(* IEC 61131-3 sources: beckhoffAutomationInterface/ST/Shark/Lib/Sequences (part 2) *)

(* ---- FB_SequenceTester.st ---- *)
(*
FB_SequenceTester — Shared test harness for sequence development.

Calls FB_SequenceOrchestrator methods directly via a REFERENCE.
Held inside a thin PROGRAM wrapper in each machine's App folder.

USAGE (thin PROGRAM wrapper pattern):
  PROGRAM PRG_SequenceTester
  VAR
      fbTester : FB_SequenceTester;
  END_VAR
      fbTester();
  // Configure: PRG_SequenceTester.Configure(refOrchestrator := PRG_Sequence.fbOrchestrator)

HOW TO TEST:
1. Set eCommand to desired command (e.g., E_Command.StartBubblerFlow)
2. Configure the corresponding parameter structure if needed
3. Set bStart := TRUE (pulse — auto-clears on rising edge)
4. Monitor sStatus, bBusy, bDone, bError, rProgress
*)
FUNCTION_BLOCK FB_SequenceTester
VAR
    // User interface — command triggers (pulse TRUE to execute)
    bStart   : BOOL;
    bStop    : BOOL;
    bReset   : BOOL;
    eCommand : E_Command := E_Command.StartBubblerFlow;

    // Parameter structures (pre-configured with realistic defaults)
    stBubblerFlowParams     : ST_CmdStartBubblerFlow := (
        side := 1,
        bubblerIndex := 1,
        flowRate := 15.0,
        hotManifoldOperatingPressure := 1.4,
        hotManifoldPressureTimeout := 600000,
        coldManifoldOperatingPressure := 1.4,
        coldManifoldPressureTimeout := 600000,
        MFCStabilizeTimeout := 60000,
        MFCFlowRateTolerance := 5.0,
        maxDepressurizingAttempts := 3
    );

    stStopBubblerFlowParams : ST_CmdStopBubblerFlow := (
        side := 1
    );

    stPurgeParams           : ST_CmdPurge := (
        mode := 1,
        side := 1,
        bubbler := 1,
        inertGasFlow := 300.0,
        purgeGasFlow := 25.0,
        purgeHighPressureLimit := 1.70,
        purgeLowPressureLimit := 0.75,
        hotManifoldOperatingPressure := 1.4,
        highPressureTimeout := 600000,
        lowPressureTimeout := 60000,
        coldManifoldPurgeCycles := 5,
        hotManifoldPurgeCycles := 5,
        purgeLinePurgeCycles := 5,
        umbilicalPurgeCycles := 5,
        umbilicalFlushTime := 60000,
        stabilisationDelay := 35000
    );

    stHeatingParams         : ST_CmdSetTemperatureGradient := (
        reactantCombiner := 60.0,
        precursorCombiner := 60.0,
        headTemp := 100.0,
        enableMode := 0
    );

    stChuckParams           : ST_CmdSetChuckZone := (
        holdSample := TRUE,
        size := 200,
        fPressureThreshold := 0.75,
        tPressureTimeout := 60000
    );

    stSpotDepositionParams  : ST_CmdSpotDeposition := (
        nDepositionCycles := 5,
        fPrecursorFlowRate := 20.0,
        fReactantFlowRate := 20.0,
        fInertMaxPurgeFlow := 250.0,
        fInertMinPurgeFlow := 100.0,
        nPrecursorBubblerIndex := 1,
        nReactantBubblerIndex := 1,
        fDistributorOperatingPressure := 2.0,
        fCombinerOperatingPressure := 1.3,
        fPressureTolerance := 5.0,
        tReactantExposureTime := 3000,
        tPrecursorExposureTime := 3000,
        tInertPurgeTime := 10000,
        tFinalPurgeTime := 30000
    );

    stLeakTestParams        : ST_CmdBubblerLeakTest := (
        side := 1,
        bubblerIndex := 1,
        leakThreshold := 0.5,
        testDuration := 300000,
        stabilizationTime := 60000,
        fillPressure := 2.5,
        testFlowRate := 20.0,
        pressureTimeout := 600000,
        pressureTolerance := 5.0,
        normalPressure := 1.4,
        depressurizeTarget := 0.5,
        normalizationFlow := 20.0
    );

    // Status output
    sStatus              : STRING(255) := 'Not configured';
    bBusy                : BOOL;
    bDone                : BOOL;
    bError               : BOOL;
    rProgress            : REAL;
    stStatus             : ST_SequenceStatus;
    stLastError          : ST_Error;
    sLastCommandResult   : STRING(255);
    bLastCommandAccepted : BOOL;

    // Debug counters
    nCycleCount   : UDINT := 0;
    nCommandCount : UDINT := 0;
    bTriggerFired : BOOL;
END_VAR
VAR
    _refOrchestrator : REFERENCE TO FB_SequenceOrchestrator;
    _bConfigured     : BOOL := FALSE;
    _rtStart         : R_TRIG;
    _rtStop          : R_TRIG;
    _rtReset         : R_TRIG;
    _sPrevStatusMsg  : STRING(255);
END_VAR

    nCycleCount   := nCycleCount + 1;
    bTriggerFired := FALSE;

    _rtStart(CLK := bStart);
    _rtStop(CLK  := bStop);
    _rtReset(CLK := bReset);

    IF NOT _bConfigured OR NOT __ISVALIDREF(_refOrchestrator) THEN
        sStatus := 'Waiting for orchestrator...';
        RETURN;
    END_IF

    IF _rtStop.Q THEN
        bStop         := FALSE;
        bTriggerFired := TRUE;
        bLastCommandAccepted := _refOrchestrator.SystemStop();
        sLastCommandResult := SEL(bLastCommandAccepted, 'SystemStop REJECTED', 'SystemStop accepted');
        nCommandCount := nCommandCount + 1;
    END_IF

    IF _rtReset.Q THEN
        bReset        := FALSE;
        bTriggerFired := TRUE;
        bLastCommandAccepted := _refOrchestrator.ErrorAcknowledge();
        sLastCommandResult := SEL(bLastCommandAccepted,
            'ErrorAcknowledge REJECTED (not in error state)',
            'ErrorAcknowledge accepted');
        nCommandCount := nCommandCount + 1;
    END_IF

    IF _rtStart.Q THEN
        bStart        := FALSE;
        bTriggerFired := TRUE;
        _ExecuteCommand();
        nCommandCount := nCommandCount + 1;
    END_IF

    stStatus    := _refOrchestrator.GetStatus();
    bBusy       := stStatus.bBusy;
    bDone       := stStatus.bDone;
    bError      := stStatus.bError;
    rProgress   := stStatus.rProgress;
    stLastError := stStatus.stLastError;

    IF bBusy THEN
        IF stStatus.sStatusMessage <> _sPrevStatusMsg THEN
            sStatus         := CONCAT('BUSY: ', stStatus.sStatusMessage);
            _sPrevStatusMsg := stStatus.sStatusMessage;
        END_IF
    ELSIF bError THEN
        IF stStatus.sStatusMessage <> _sPrevStatusMsg THEN
            sStatus         := CONCAT('ERROR: ', stStatus.sStatusMessage);
            _sPrevStatusMsg := stStatus.sStatusMessage;
        END_IF
    ELSIF bDone THEN
        IF stStatus.sStatusMessage <> _sPrevStatusMsg THEN
            sStatus         := CONCAT('DONE: ', stStatus.sStatusMessage);
            _sPrevStatusMsg := stStatus.sStatusMessage;
        END_IF
    ELSE
        sStatus         := SEL(sLastCommandResult = '', 'Ready', sLastCommandResult);
        _sPrevStatusMsg := '';
    END_IF

END_FUNCTION_BLOCK

// =============================================================================
// PUBLIC API
// =============================================================================

METHOD PUBLIC Configure : BOOL
VAR_INPUT
    refOrchestrator : REFERENCE TO FB_SequenceOrchestrator;
END_VAR
    IF NOT __ISVALIDREF(refOrchestrator) THEN RETURN; END_IF
    _refOrchestrator REF= refOrchestrator;
    _bConfigured     := TRUE;
    sStatus          := 'Ready';
    sLastCommandResult := '';
    Configure        := TRUE;
END_METHOD

// =============================================================================
// PRIVATE
// =============================================================================

METHOD PRIVATE _ExecuteCommand
VAR
    bSuccess      : BOOL;
    stHoldParams  : ST_ChuckVacuumHold;
    stReleaseParams : ST_ChuckVacuumRelease;
END_VAR
    bSuccess             := FALSE;
    bLastCommandAccepted := FALSE;

    CASE eCommand OF
        E_Command.StartBubblerFlow:
            bSuccess := _refOrchestrator.StartBubblerFlow(stBubblerFlowParams);
            sLastCommandResult := SEL(bSuccess,
                'StartBubblerFlow REJECTED (sequence busy or in error)',
                'StartBubblerFlow accepted');

        E_Command.StopBubblerFlow:
            bSuccess := _refOrchestrator.StopBubblerFlow(stStopBubblerFlowParams);
            sLastCommandResult := SEL(bSuccess, 'StopBubblerFlow REJECTED', 'StopBubblerFlow accepted');

        E_Command.StartPurge:
            bSuccess := _refOrchestrator.StartPurge(stPurgeParams);
            sLastCommandResult := SEL(bSuccess, 'StartPurge REJECTED', 'StartPurge accepted');

        E_Command.SetTemperatureGradients:
            bSuccess := _refOrchestrator.StartHeating(stHeatingParams);
            sLastCommandResult := SEL(bSuccess, 'StartHeating REJECTED', 'StartHeating accepted');

        E_Command.HoldReleaseSample:
            IF stChuckParams.holdSample THEN
                stHoldParams.iSelectZone            := _WaferSizeToZoneCount(stChuckParams.size);
                stHoldParams.fLockPressureThreshold := stChuckParams.fPressureThreshold;
                stHoldParams.tPressureTimeout       := DINT_TO_TIME(stChuckParams.tPressureTimeout);
                bSuccess := _refOrchestrator.StartChuckVacuumHold(stHoldParams);
                sLastCommandResult := SEL(bSuccess, 'ChuckVacuumHold REJECTED', 'ChuckVacuumHold accepted');
            ELSE
                stReleaseParams.fReleasePressureThreshold := stChuckParams.fPressureThreshold;
                stReleaseParams.tPressureTimeout          := DINT_TO_TIME(stChuckParams.tPressureTimeout);
                bSuccess := _refOrchestrator.StartChuckVacuumRelease(stReleaseParams);
                sLastCommandResult := SEL(bSuccess, 'ChuckVacuumRelease REJECTED', 'ChuckVacuumRelease accepted');
            END_IF

        E_Command.CancelProcess:
            bSuccess := _refOrchestrator.SystemStop();
            sLastCommandResult := SEL(bSuccess, 'SystemStop REJECTED', 'SystemStop accepted');

        E_Command.ErrorAcknowledge:
            bSuccess := _refOrchestrator.ErrorAcknowledge();
            sLastCommandResult := SEL(bSuccess,
                'ErrorAcknowledge REJECTED (not in error state)',
                'ErrorAcknowledge accepted');

        E_Command.StartSpotDeposition:
            bSuccess := _refOrchestrator.StartSpotDeposition(stSpotDepositionParams);
            sLastCommandResult := SEL(bSuccess, 'SpotDeposition REJECTED', 'SpotDeposition accepted');

        E_Command.StartBubblerLeakTest:
            bSuccess := _refOrchestrator.StartBubblerLeakTest(stLeakTestParams);
            sLastCommandResult := SEL(bSuccess, 'BubblerLeakTest REJECTED', 'BubblerLeakTest accepted');

        E_Command.None:
            sLastCommandResult := 'No command selected (eCommand = None)';

    ELSE
        sLastCommandResult := 'Unknown command';
    END_CASE

    bLastCommandAccepted := bSuccess;
END_METHOD

METHOD PRIVATE _WaferSizeToZoneCount : INT
VAR_INPUT
    nWaferSize : INT;
END_VAR
    IF nWaferSize <= 150 THEN
        _WaferSizeToZoneCount := 1;
    ELSIF nWaferSize <= 200 THEN
        _WaferSizeToZoneCount := 2;
    ELSE
        _WaferSizeToZoneCount := 3;
    END_IF
END_METHOD

(* ---- FB_SpotDepositionSequence.st ---- *)
(*
FB_SpotDepositionSequence
ALD spot deposition cycle: alternating precursor/reactant exposures
separated by inert gas purges.

CYCLE STRUCTURE (per deposition cycle):
  Inert Purge -> Reactant Exposure -> Inert Purge -> Precursor Exposure

FULL SEQUENCE:
  1. Init:       Prepare exhaust vacuum
  2. Startup A:  Start precursor gas (A-Side) via FB_GasStartSequence
  3. Startup B:  Start reactant gas (B-Side) via FB_GasStartSequence
  4. Cycles:     N x (InertPurge -> ReactantExpose -> InertPurge -> PrecursorExpose)
  5. FinalPurge: Extended inert purge to clear lines
  6. Shutdown:   Stop both sides via FB_GasStopSequence

HARDWARE:
  - A-Side: Precursor MFC + bubbler + valves
  - B-Side: Reactant MFC + bubbler + valves
  - Inert:  IG MFC + inert gas valve (purge between exposures)
  - Common: Exhaust pump, nozzle (start) valves
*)
FUNCTION_BLOCK FB_SpotDepositionSequence IMPLEMENTS I_TreeNode
VAR
    // Internal State
    _bInitialized    : BOOL := FALSE;
    _bParamsConfigured : BOOL := FALSE;
    _ePhase          : INT := 0;

    // Sub-sequences
    _fbPrepareExhaust  : FB_PrepareExhaustSequence;
    _fbGasStartA       : FB_GasStartSequence;
    _fbGasStartB       : FB_GasStartSequence;
    _fbGasStopA        : FB_GasStopSequence;
    _fbGasStopB        : FB_GasStopSequence;

    // Inert gas hardware
    _ipInertValve      : I_Valve;
    _ipInertMFC        : I_Controller;
    _ipNozzleA         : I_Valve;
    _ipNozzleB         : I_Valve;

    // Cycle tracking
    _nCurrentCycle     : DINT;
    _nCycleSubPhase    : INT;

    // Parameters
    _stParams          : ST_CmdSpotDeposition;

    // Timing
    _fbTimer           : TON;

    // Status
    _bError            : BOOL;
    _sErrorMsg         : STRING(255);
END_VAR

VAR CONSTANT
    PHASE_IDLE           : INT := 0;
    PHASE_INIT           : INT := 1;
    PHASE_STARTUP_A      : INT := 2;
    PHASE_STARTUP_B      : INT := 3;
    PHASE_CYCLES         : INT := 4;
    PHASE_FINAL_PURGE    : INT := 5;
    PHASE_SHUTDOWN       : INT := 6;
    PHASE_DONE           : INT := 7;
    PHASE_ERROR          : INT := 99;

    SUB_INERT_PURGE_1    : INT := 0;
    SUB_REACTANT_EXPOSE  : INT := 1;
    SUB_INERT_PURGE_2    : INT := 2;
    SUB_PRECURSOR_EXPOSE : INT := 3;
END_VAR

METHOD PUBLIC Init : BOOL
VAR_INPUT
    ipProvider : I_HardwareProvider;
END_VAR
    _bInitialized := FALSE;
    _bParamsConfigured := FALSE;
    _ePhase := PHASE_IDLE;
    _bError := FALSE;
    _sErrorMsg := '';

    IF ipProvider = 0 THEN
        GVL_ErrorLogger.Logger.LogError('FB_SpotDepositionSequence', E_ErrorId.ERR_GEN_NULL_POINTER, 'Provider is null');
        RETURN;
    END_IF

    IF NOT _fbPrepareExhaust.Init(ipProvider, E_GasSide.A_SIDE) THEN RETURN; END_IF
    IF NOT _fbGasStartA.Init(ipProvider := ipProvider, eSide := E_GasSide.A_SIDE) THEN RETURN; END_IF
    IF NOT _fbGasStartB.Init(ipProvider := ipProvider, eSide := E_GasSide.B_SIDE) THEN RETURN; END_IF
    IF NOT _fbGasStopA.Init(ipProvider := ipProvider, eSide := E_GasSide.A_SIDE) THEN RETURN; END_IF
    IF NOT _fbGasStopB.Init(ipProvider := ipProvider, eSide := E_GasSide.B_SIDE) THEN RETURN; END_IF

    _ipInertValve := ipProvider.GetInertGasValve();
    _ipInertMFC := ipProvider.GetInertMFCController();
    _ipNozzleA := ipProvider.GetNozzleIsoValve(E_GasSide.A_SIDE);
    _ipNozzleB := ipProvider.GetNozzleIsoValve(E_GasSide.B_SIDE);

    IF _ipInertValve = 0 OR _ipInertMFC = 0 OR _ipNozzleA = 0 OR _ipNozzleB = 0 THEN
        GVL_ErrorLogger.Logger.LogError('FB_SpotDepositionSequence', E_ErrorId.ERR_GEN_NULL_POINTER, 'Inert gas or nozzle hardware not found');
        RETURN;
    END_IF

    _bInitialized := TRUE;
    Init := TRUE;
END_METHOD

METHOD PUBLIC SetParams
VAR_INPUT
    stParams : ST_CmdSpotDeposition;
END_VAR
VAR
    stStartA : ST_CmdStartBubblerFlow;
    stStartB : ST_CmdStartBubblerFlow;
END_VAR
    IF NOT _bInitialized THEN RETURN; END_IF

    _stParams := stParams;

    stStartA.flowRate := stParams.fPrecursorFlowRate;
    stStartA.bubblerIndex := DINT_TO_INT(stParams.nPrecursorBubblerIndex);
    stStartA.coldManifoldOperatingPressure := stParams.fDistributorOperatingPressure;
    stStartA.hotManifoldOperatingPressure := stParams.fCombinerOperatingPressure;
    stStartA.MFCFlowRateTolerance := stParams.fPressureTolerance;
    _fbGasStartA.SetParams(stStartA);

    stStartB.flowRate := stParams.fReactantFlowRate;
    stStartB.bubblerIndex := DINT_TO_INT(stParams.nReactantBubblerIndex);
    stStartB.coldManifoldOperatingPressure := stParams.fDistributorOperatingPressure;
    stStartB.hotManifoldOperatingPressure := stParams.fCombinerOperatingPressure;
    stStartB.MFCFlowRateTolerance := stParams.fPressureTolerance;
    _fbGasStartB.SetParams(stStartB);
    _bParamsConfigured := TRUE;
END_METHOD

METHOD PUBLIC Tick : ST_NodeResult
VAR
    stResult : ST_NodeResult;
END_VAR
    IF NOT _bInitialized THEN
        Tick.eStatus := E_NodeStatus.FAILURE;
        Tick.bHasError := TRUE;
        Tick.stError.eErrorId := E_ErrorId.ERR_GEN_INITIALIZATION;
        Tick.stError.sSource := 'FB_SpotDepositionSequence';
        Tick.stError.sMessage := 'Init must be called before Tick';
        Tick.sDescription := Tick.stError.sMessage;
        RETURN;
    END_IF

    IF NOT _bParamsConfigured THEN
        Tick.eStatus := E_NodeStatus.FAILURE;
        Tick.bHasError := TRUE;
        Tick.stError.eErrorId := E_ErrorId.ERR_GEN_NOT_CONFIGURED;
        Tick.stError.sSource := 'FB_SpotDepositionSequence';
        Tick.stError.sMessage := 'SetParams must be called before Tick';
        Tick.sDescription := Tick.stError.sMessage;
        RETURN;
    END_IF

    CASE _ePhase OF
        PHASE_IDLE:
            _ePhase := PHASE_INIT;
            _fbPrepareExhaust.Reset();

        PHASE_INIT:
            stResult := _fbPrepareExhaust.Tick();
            IF stResult.eStatus = E_NodeStatus.SUCCESS THEN
                _fbGasStartA.Reset();
                _ePhase := PHASE_STARTUP_A;
            ELSIF stResult.eStatus = E_NodeStatus.FAILURE THEN
                _SetError('Exhaust preparation failed');
            END_IF

        PHASE_STARTUP_A:
            stResult := _fbGasStartA.Tick();
            IF stResult.eStatus = E_NodeStatus.SUCCESS THEN
                _fbGasStartB.Reset();
                _ePhase := PHASE_STARTUP_B;
            ELSIF stResult.eStatus = E_NodeStatus.FAILURE THEN
                _SetError('Precursor gas start failed');
            END_IF

        PHASE_STARTUP_B:
            stResult := _fbGasStartB.Tick();
            IF stResult.eStatus = E_NodeStatus.SUCCESS THEN
                _nCurrentCycle := 1;
                _nCycleSubPhase := SUB_INERT_PURGE_1;
                _fbTimer(IN := FALSE);
                _ePhase := PHASE_CYCLES;
            ELSIF stResult.eStatus = E_NodeStatus.FAILURE THEN
                _SetError('Reactant gas start failed');
            END_IF

        PHASE_CYCLES:
            _ExecuteCycle();

        PHASE_FINAL_PURGE:
            _fbTimer(IN := TRUE, PT := DINT_TO_TIME(_stParams.tFinalPurgeTime));
            IF _fbTimer.Q THEN
                _ipInertMFC.SetSetpoint(0.0);
                _ipInertValve.Close();
                _fbGasStopA.Reset();
                _fbGasStopB.Reset();
                _ePhase := PHASE_SHUTDOWN;
            END_IF

        PHASE_SHUTDOWN:
            stResult := _fbGasStopA.Tick();
            IF stResult.eStatus = E_NodeStatus.SUCCESS THEN
                stResult := _fbGasStopB.Tick();
                IF stResult.eStatus = E_NodeStatus.SUCCESS THEN
                    _ePhase := PHASE_DONE;
                ELSIF stResult.eStatus = E_NodeStatus.FAILURE THEN
                    _SetError('B-Side gas stop failed');
                END_IF
            ELSIF stResult.eStatus = E_NodeStatus.FAILURE THEN
                _SetError('A-Side gas stop failed');
            ELSE
                _fbGasStopB.Tick();
            END_IF

        PHASE_DONE:
            ;

        PHASE_ERROR:
            ;
    END_CASE

    IF _ePhase = PHASE_DONE THEN
        Tick.eStatus := E_NodeStatus.SUCCESS;
        Tick.rProgress := 100.0;
        Tick.sDescription := 'Spot Deposition Complete';
    ELSIF _ePhase = PHASE_ERROR THEN
        Tick.eStatus := E_NodeStatus.FAILURE;
        Tick.bHasError := TRUE;
        Tick.stError.eErrorId := E_ErrorId.ERR_GEN_INTERNAL;
        Tick.stError.sSource := 'FB_SpotDepositionSequence';
        Tick.stError.sMessage := _sErrorMsg;
        Tick.sDescription := _sErrorMsg;
    ELSE
        Tick.eStatus := E_NodeStatus.RUNNING;
        Tick.sDescription := CONCAT('Spot Deposition: Phase ', INT_TO_STRING(_ePhase));
        IF _ePhase = PHASE_CYCLES AND _stParams.nDepositionCycles > 0 THEN
            Tick.rProgress := 10.0 + TO_REAL((DINT_TO_LREAL(_nCurrentCycle - 1) / DINT_TO_LREAL(_stParams.nDepositionCycles)) * 80.0);
        END_IF
    END_IF
END_METHOD

METHOD PRIVATE _ExecuteCycle
    CASE _nCycleSubPhase OF
        SUB_INERT_PURGE_1, SUB_INERT_PURGE_2:
            IF NOT _fbTimer.IN THEN
                _ipNozzleA.Close();
                _ipNozzleB.Close();
                _ipInertValve.Open();
                _ipInertMFC.SetSetpoint(REAL_TO_LREAL(_stParams.fInertMaxPurgeFlow));
            END_IF
            _fbTimer(IN := TRUE, PT := DINT_TO_TIME(_stParams.tInertPurgeTime));
            IF _fbTimer.Q THEN
                _fbTimer(IN := FALSE);
                _ipInertMFC.SetSetpoint(REAL_TO_LREAL(_stParams.fInertMinPurgeFlow));
                _ipInertValve.Close();
                _nCycleSubPhase := _nCycleSubPhase + 1;
            END_IF

        SUB_REACTANT_EXPOSE:
            IF NOT _fbTimer.IN THEN
                _ipNozzleB.Open();
            END_IF
            _fbTimer(IN := TRUE, PT := DINT_TO_TIME(_stParams.tReactantExposureTime));
            IF _fbTimer.Q THEN
                _fbTimer(IN := FALSE);
                _ipNozzleB.Close();
                _nCycleSubPhase := _nCycleSubPhase + 1;
            END_IF

        SUB_PRECURSOR_EXPOSE:
            IF NOT _fbTimer.IN THEN
                _ipNozzleA.Open();
            END_IF
            _fbTimer(IN := TRUE, PT := DINT_TO_TIME(_stParams.tPrecursorExposureTime));
            IF _fbTimer.Q THEN
                _fbTimer(IN := FALSE);
                _ipNozzleA.Close();
                _nCurrentCycle := _nCurrentCycle + 1;
                IF _nCurrentCycle > _stParams.nDepositionCycles THEN
                    _ipInertValve.Open();
                    _ipInertMFC.SetSetpoint(REAL_TO_LREAL(_stParams.fInertMaxPurgeFlow));
                    _fbTimer(IN := FALSE);
                    _ePhase := PHASE_FINAL_PURGE;
                ELSE
                    _nCycleSubPhase := SUB_INERT_PURGE_1;
                END_IF
            END_IF
    END_CASE
END_METHOD

METHOD PRIVATE _SetError
VAR_INPUT
    sMsg : STRING(255);
END_VAR
    _sErrorMsg := sMsg;
    _bError := TRUE;
    _ePhase := PHASE_ERROR;
END_METHOD

METHOD PUBLIC Reset : BOOL
    _ePhase := PHASE_IDLE;
    _bError := FALSE;
    _sErrorMsg := '';
    _nCurrentCycle := 0;
    _nCycleSubPhase := 0;
    _fbTimer(IN := FALSE);
    _fbPrepareExhaust.Reset();
    _fbGasStartA.Reset();
    _fbGasStartB.Reset();
    _fbGasStopA.Reset();
    _fbGasStopB.Reset();
    Reset := TRUE;
END_METHOD

METHOD PUBLIC Halt
    IF _ipInertMFC <> 0 THEN _ipInertMFC.SetSetpoint(0.0); END_IF
    IF _ipInertValve <> 0 THEN _ipInertValve.Close(); END_IF
    IF _ipNozzleA <> 0 THEN _ipNozzleA.Close(); END_IF
    IF _ipNozzleB <> 0 THEN _ipNozzleB.Close(); END_IF
    _fbGasStopA.Halt();
    _fbGasStopB.Halt();
    Reset();
END_METHOD

PROPERTY PUBLIC NodeName : STRING(50)
    GET
        NodeName := 'SpotDeposition';
    END_GET
END_PROPERTY

END_FUNCTION_BLOCK

(* ---- FB_SystemStopSequence.st ---- *)
(*
FB_SystemStopSequence
Parallel gas shutdown of both sides + exhaust isolation.
*)
FUNCTION_BLOCK FB_SystemStopSequence IMPLEMENTS I_TreeNode
VAR
    _seq : FB_SequenceNode;
    // Parallel gas shutdown (both sides)
    stepParallelGasStop : FB_ParallelNode;
    stepGasStopA         : FB_GasStopSequence;
    stepGasStopB         : FB_GasStopSequence;

    // Exhaust shutdown
    stepCloseExhaustVacuumIso : FB_CloseValveNode;

    // Internal state
    _bInitialized    : BOOL := FALSE;
END_VAR

METHOD PUBLIC Init : BOOL
VAR_INPUT
    ipProvider : I_HardwareProvider;
END_VAR
VAR
    ipExhaustVacuumIsoValve : I_Valve;
END_VAR
    IF _bInitialized THEN
        Init := TRUE;
        RETURN;
    END_IF

    IF ipProvider = 0 THEN
        GVL_ErrorLogger.Logger.LogError('FB_SystemStopSequence', E_ErrorId.ERR_GEN_NULL_POINTER, 'Provider is null');
        RETURN;
    END_IF

    // Parallel gas shutdown (A and B sides simultaneously)
    stepGasStopA.Init(ipProvider := ipProvider, eSide := E_GasSide.A_SIDE);
    stepGasStopA.NodeName := 'GasStop_A';

    stepGasStopB.Init(ipProvider := ipProvider, eSide := E_GasSide.B_SIDE);
    stepGasStopB.NodeName := 'GasStop_B';

    stepParallelGasStop.AddChild(stepGasStopA);
    stepParallelGasStop.AddChild(stepGasStopB);
    stepParallelGasStop.sName := 'ParallelGasStop';
    _seq.AddChild(stepParallelGasStop);

    // Exhaust shutdown
    ipExhaustVacuumIsoValve := ipProvider.GetExhaustVacuumIsoValve();
    stepCloseExhaustVacuumIso.Init(ipExhaustVacuumIsoValve, sNodeName := 'CloseExhaustVacuumIso');
    _seq.AddChild(stepCloseExhaustVacuumIso);

    _seq.sName := 'SystemStop';

    _bInitialized := TRUE;
    Init := TRUE;
END_METHOD

PROPERTY PUBLIC NodeName : STRING(50)
    GET
        NodeName := _seq.sName;
    END_GET
    SET
        _seq.sName := NodeName;
    END_SET
END_PROPERTY

METHOD Tick : ST_NodeResult
    IF NOT _bInitialized THEN
        Tick.eStatus := E_NodeStatus.FAILURE;
        Tick.bHasError := TRUE;
        Tick.stError.eErrorId := E_ErrorId.ERR_GEN_INITIALIZATION;
        Tick.stError.sSource := 'FB_SystemStopSequence';
        Tick.stError.sMessage := 'Init must be called before Tick';
        Tick.sDescription := Tick.stError.sMessage;
        RETURN;
    END_IF

    Tick := _seq.Tick();
END_METHOD

{attribute 'estimated-stack-usage' := '500'}
METHOD Reset : BOOL
    Reset := _seq.Reset();
END_METHOD

{attribute 'estimated-stack-usage' := '500'}
METHOD Halt
    _seq.Halt();
END_METHOD

END_FUNCTION_BLOCK
